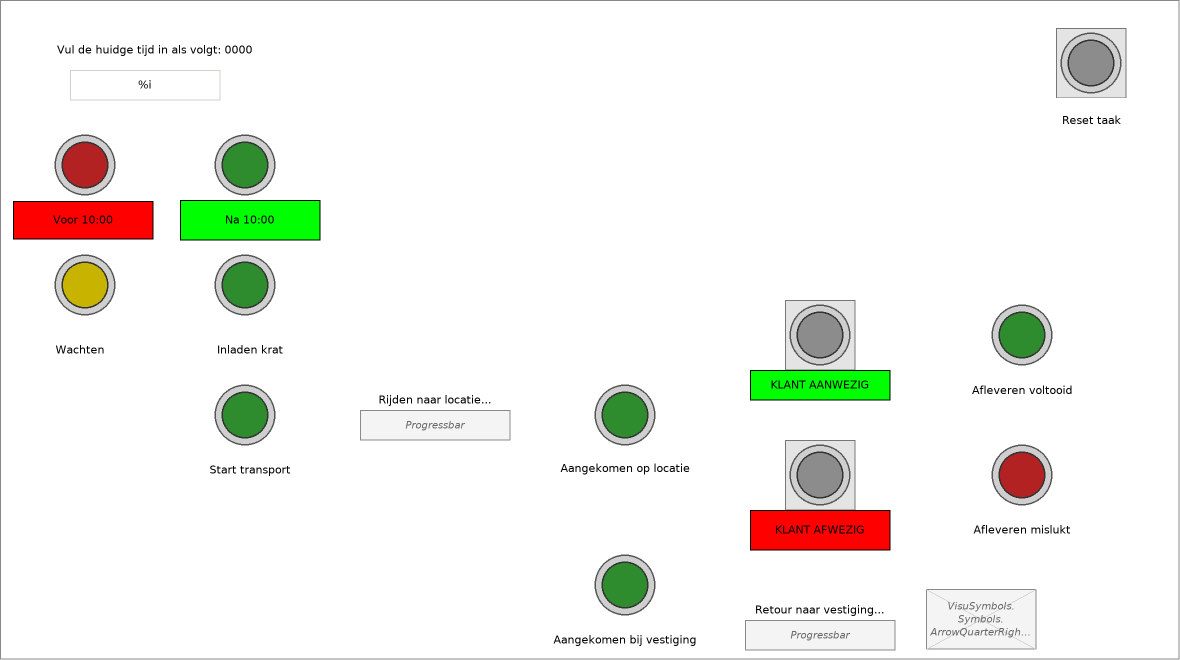
VISUALIZATION Transporteren_order  // 1180x660
    Rectangle (745,590 150x40), "Retour naar vestiging..."
    Rectangle (360,380 150x40), "Rijden naar locatie..."
    Label (40,30 230x40), "Vul de huidge tijd in als volgt: 0000"
    Textfield (70,70 150x30), "%i", text variable: Transporteren_order.Huidige_tijd
        OnMouseClick: write the text variable via Default, min 0, max 2400
    Lamp1 (50,130 70x70), variable: Transporteren_order.Voor10Uur, style: Lamp-Lamp1-Red
    Lamp1 (210,130 70x70), variable: Transporteren_order.Na10Uur, style: Lamp-Lamp1-Green
    Rectangle (13,201 140x38), "Voor 10:00"
    Rectangle (180,200 140x40), "Na 10:00"
    Lamp1 (50,250 70x70), variable: Transporteren_order.Wachten, style: Lamp-Lamp1-Yellow
    Rectangle (20,330 120x40), "Wachten"
    Lamp1 (210,250 70x70), variable: Transporteren_order.Inladen_krat, style: Lamp-Lamp1-Green
    Rectangle (190,330 120x40), "Inladen krat"
    Rectangle (190,450 120x40), "Start transport"
    Lamp1 (210,380 70x70), variable: Transporteren_order.Start_transport, style: Lamp-Lamp1-Green
    Progressbar (360,410 150x30), variable: Transporteren_order.WachtTijd_1
    Rectangle (509,446 233x45), "Aangekomen op locatie"
    Lamp1 (590,380 70x70), variable: Transporteren_order.Locatie, style: Lamp-Lamp1-Green
    PushSwitch (785,300 70x70), variable: Transporteren_order.Klant_aanwezig, behaviour: TOGGLE, style: Switch-PushSwitch-Gray
    Rectangle (750,370 140x30), "KLANT AANWEZIG"
    PushSwitch (785,440 70x70), variable: Transporteren_order.Klant_afwezig, behaviour: TOGGLE, style: Switch-PushSwitch-Gray
    Rectangle (750,510 140x40), "KLANT AFWEZIG"
    Rectangle (906,368 233x45), "Afleveren voltooid"
    Lamp1 (987,300 70x70), variable: Transporteren_order.Afleveren_voltooid, style: Lamp-Lamp1-Green
    Rectangle (907,510 230x40), "Afleveren mislukt"
    Lamp1 (987,440 70x70), variable: Transporteren_order.Afleveren_mislukt, style: Lamp-Lamp1-Red
    Image (926,589 110x60), image: VisuSymbols.Symbols.ArrowQuarterRightLeft
    Progressbar (745,620 150x30), variable: Transporteren_order.WachtTijd_2
    Lamp1 (590,550 70x70), variable: Transporteren_order.Retour_vestiging, style: Lamp-Lamp1-Green
    Rectangle (510,620 230x40), "Aangekomen bij vestiging"
    PushSwitch (1056,28 70x70), variable: Transporteren_order.Taak2Reset, behaviour: TAP, style: Switch-PushSwitch-Gray
    Rectangle (1003,98 177x45), "Reset taak"
END_VISUALIZATION

(* stored: Version 1.1.0.1, ProductVersion 3.1.4024.12
   Visu Transporteren_order: Id {bcb93648-7631-4be5-8f1c-4affd6897e2e} *)
